FUNCTION_BLOCK T_RoboConnect_SetToolDigitalOutput_CorrectIndexPasses EXTENDS T_UnitTestBase
VAR
  robot : I_RoboConnect;
  targetDO : UINT;
  myTestState, prevState :
    (INIT, ARRANGE, ACT, ASSERT) := INIT;
  expected, actual : BOOL;
  counter : UINT;
END_VAR

CASE myTestState OF
  INIT:
    StateChanged();
    myTestState := ARRANGE;

  ARRANGE:
    IF StateChanged() THEN
      expected := TRUE;
      myTestState := ACT;
    END_IF

  ACT:
    actual := robot.SetToolDigitalOutput(targetDO, TRUE);
    myTestState := ASSERT;

  ASSERT:
    assertion.AssertEquals_BOOL(expected, actual, 'robot.GetDigitalOutput(targetDO) := TRUE');
    TestFinished();
    myTestState := INIT;

END_CASE

METHOD FB_init : BOOL
VAR_INPUT
  bInitRetains : BOOL; // if TRUE, the retain variables are initialized (warm start / cold start)
  bInCopyCode : BOOL; // if TRUE, the instance afterwards gets moved into the copy code (online change)
  TestSuite : tcl_SimpleUnitTestLibrary.I_TestSuite;
  robot : I_TcRobot;
  targetDo : UINT;
END_VAR
THIS^.robot := robot;
THIS^.targetDo := targetDo;
END_METHOD

METHOD PRIVATE StateChanged : BOOL
IF  myTestState = prevState THEN
  RETURN;
END_IF

prevState := myTestState;
StateChanged := TRUE;
END_METHOD

METHOD WaitForCycles : BOOL
VAR_INPUT
  maxCount : UINT;
END_VAR
counter := counter + 1;

IF counter = maxCount THEN
  counter := 0;
  WaitForCycles := TRUE;
END_IF
END_METHOD

END_FUNCTION_BLOCK

(* stored: Version 1.1.0.1
   POU T_TcRobot_SetToolDigitalOutput_CorrectIndexPasses: Id {23f4c917-2de2-426f-8772-55791dd30636}, SpecialFunc None
   Method FB_init: Id {a94e2146-bc27-47e6-9705-ce0c31b0c4a5}
   Method StateChanged: Id {53fdeac1-afcc-4aa3-9529-7691e2b4616b}
   Method WaitForCycles: Id {b8f41076-dbdc-42aa-b817-5761c9f251b7} *)
